                   IF #Minuty < 10 THEN
                       #StrMin := CONCAT(IN1 := '0', IN2 := #StrMin);
                   END_IF;
                   IF #Sekundy < 10 THEN
                       #StrSec := CONCAT(IN1 := '0', IN2 := #StrSec);
                   END_IF;

                   IF "DB_Data".Stanowisko1."Time".RemainingSec <= 0 AND "DB_Data".Stanowisko1."Time".Blink THEN
                       "DB_Data".Stanowisko1."Time".RemainingStr := '     ';
                   ELSE
                       "DB_Data".Stanowisko1."Time".RemainingStr := CONCAT(IN1 := #StrMin, IN2 := CONCAT(IN1 := ':', IN2 := #StrSec));
                   END_IF;

           END_CASE;

           //Przejscie do stanu awarii
           IF "DB_Data".Stanowisko1.Commands.ReportFault.State THEN
               "DB_Data".Stanowisko1.Production.State := 3;
               "DB_Data".Stanowisko1.Commands.ReportFault.State := 0;
           END_IF;

           //Przejscie do zakonczenia montazu
           IF "DB_Data".Stanowisko1.Commands.FInish.State THEN
               "DB_Data".Stanowisko1.Production.State := 2;
               "DB_Data".Stanowisko1.Commands.FInish.State := 0;
           END_IF;

       2:
           //Ustawienie przycisków
           "DB_Data".Stanowisko1.Commands.Start.Enable := 0;
           "DB_Data".Stanowisko1.Commands.AbortProcess.Enable := 0;
           "DB_Data".Stanowisko1.Commands.FInish.Enable := 0;
           "DB_Data".Stanowisko1.Commands.ReportFault.Enable := 0;

           #temp_start_time := RD_LOC_T(OUT => "DB_Zlecenia".NastepneZlecenie.Zlecenie."Time".Stanowisko1.EndTime); // Zapis czasu zakonczenia

           //Funkcja zapisujaca wyrob do bazy danych dla innych stanowisk
           FOR #i := 0 TO 199 DO

               // szukanie pierwszego wolnego miejsca (czyli takiego, gdzie ID zlecenia to 0)
               IF "DB_Zlecenia".Zlecenie[#i].Zlecenie.ID = 0 THEN

                   "DB_Zlecenia".Zlecenie[#i] := "DB_Zlecenia".NastepneZlecenie;

                   //Status stanowiska 1 - praca zakonczona
                   "DB_Zlecenia".Zlecenie[#i].Zlecenie.Status[0] := TRUE;

                   //Obliczenie faktycznego czasu pracy (sekundy, zaokraglone)
                   #temp_diff_time := "DB_Zlecenia".Zlecenie[#i].Zlecenie."Time".Stanowisko1.EndTime - "DB_Zlecenia".Zlecenie[#i].Zlecenie."Time".Stanowisko1.StartTime;
                   "DB_Zlecenia".Zlecenie[#i].Zlecenie."Time".Stanowisko1.ActualTime := DINT_TO_INT((TIME_TO_DINT(#temp_diff_time) + 500) / 1000);

                   //Jesli zlecenie mialo wiecej niz 1 sztuke - zostaw ID/Model, zmniejsz PartNo, wyczysc Time/Alarm
                   IF "DB_Zlecenia".NastepneZlecenie.Zlecenie.PartNo > 1 THEN
                       "DB_Zlecenia".NastepneZlecenie.Zlecenie.PartNo := "DB_Zlecenia".NastepneZlecenie.Zlecenie.PartNo - 1;
                       "DB_Zlecenia".NastepneZlecenie.Zlecenie."Time" := "DB_Zlecenia".PusteZlecenie.Zlecenie."Time";
                       "DB_Zlecenia".NastepneZlecenie.Zlecenie.Alarm := "DB_Zlecenia".PusteZlecenie.Zlecenie.Alarm;
                   ELSE
                       "DB_Zlecenia".NastepneZlecenie := "DB_Zlecenia".PusteZlecenie;
                   END_IF;
                   EXIT;
               END_IF;
           END_FOR;

           "DB_Data".Stanowisko1.Stats.DoneToday := "DB_Data".Stanowisko1.Stats.DoneToday + 1;
           "DB_Data".DoneAllTime[0] := "DB_Data".DoneAllTime[0] + 1;

           "DB_Data".Stanowisko1.Production.State := 0;
       3:
           //Ustawienie przycisków
           "DB_Data".Stanowisko1.Commands.Start.Enable := 0;
           "DB_Data".Stanowisko1.Commands.AbortProcess.Enable := 1;
           "DB_Data".Stanowisko1.Commands.FInish.Enable := 0;
           "DB_Data".Stanowisko1.Commands.ReportFault.Enable := 0;

           //Dodanie alarmow
           "DB_Zlecenia".NastepneZlecenie.Zlecenie.Alarm.Stanowisko1 := "DB_Data".Stanowisko1.Commands.FaultReason;

           IF "DB_Data".Stanowisko1.Commands.AbortProcess.State THEN
               #temp_start_time := RD_LOC_T(OUT => "DB_Zlecenia".NastepneZlecenie.Zlecenie."Time".Stanowisko1.EndTime); // Zapis czasu zakonczenia

               //Funkcja zapisujaca wyrob do bazy danych dla innych stanowisk
               FOR #i := 0 TO 199 DO
                   IF "DB_Zlecenia".Zlecenie[#i].Zlecenie.ID = 0 THEN

                       "DB_Zlecenia".Zlecenie[#i] := "DB_Zlecenia".NastepneZlecenie;
                       "DB_Zlecenia".Zlecenie[#i].Zlecenie."Time".Stanowisko1.Abort := TRUE;

                       //Status stanowiska 1 - praca zakonczona (przez abort)
                       "DB_Zlecenia".Zlecenie[#i].Zlecenie.Status[0] := TRUE;

                       //Obliczenie faktycznego czasu pracy (sekundy, zaokraglone)
                       #temp_diff_time := "DB_Zlecenia".Zlecenie[#i].Zlecenie."Time".Stanowisko1.EndTime - "DB_Zlecenia".Zlecenie[#i].Zlecenie."Time".Stanowisko1.StartTime;
                       "DB_Zlecenia".Zlecenie[#i].Zlecenie."Time".Stanowisko1.ActualTime := DINT_TO_INT((TIME_TO_DINT(#temp_diff_time) + 500) / 1000);

                       IF "DB_Zlecenia".NastepneZlecenie.Zlecenie.PartNo > 1 THEN
                           "DB_Zlecenia".NastepneZlecenie.Zlecenie.PartNo := "DB_Zlecenia".NastepneZlecenie.Zlecenie.PartNo - 1;
                           "DB_Zlecenia".NastepneZlecenie.Zlecenie."Time" := "DB_Zlecenia".PusteZlecenie.Zlecenie."Time";
                           "DB_Zlecenia".NastepneZlecenie.Zlecenie.Alarm := "DB_Zlecenia".PusteZlecenie.Zlecenie.Alarm;
                       ELSE
                           "DB_Zlecenia".NastepneZlecenie := "DB_Zlecenia".PusteZlecenie;
                       END_IF;

                       "DB_Data".Stanowisko1.Commands.AbortProcess.State := 0;
                       "DB_Data".Stanowisko1.Production.State := 0;
                       EXIT;
                   END_IF;
               END_FOR;
           END_IF;

   END_CASE;
   IF "DB_Data".Stanowisko1.Commands.AbortProcess.State THEN
       "DB_Data".Stanowisko1.Production.State := 0;
       "DB_Data".Stanowisko1.Commands.AbortProcess.State := 0;

       #temp_start_time := RD_LOC_T(OUT => "DB_Zlecenia".NastepneZlecenie.Zlecenie."Time".Stanowisko1.EndTime); // Zapis czasu zakonczenia

       //Funkcja zapisujaca wyrob do bazy danych dla innych stanowisk
       FOR #i := 0 TO 199 DO
           IF "DB_Zlecenia".Zlecenie[#i].Zlecenie.ID = 0 THEN

               "DB_Zlecenia".Zlecenie[#i] := "DB_Zlecenia".NastepneZlecenie;
               "DB_Zlecenia".Zlecenie[#i].Zlecenie."Time".Stanowisko1.Abort := TRUE;

               //Status stanowiska 1 - praca zakonczona (przez abort)
               "DB_Zlecenia".Zlecenie[#i].Zlecenie.Status[0] := TRUE;

               //Obliczenie faktycznego czasu pracy (sekundy, zaokraglone)
               #temp_diff_time := "DB_Zlecenia".Zlecenie[#i].Zlecenie."Time".Stanowisko1.EndTime - "DB_Zlecenia".Zlecenie[#i].Zlecenie."Time".Stanowisko1.StartTime;
               "DB_Zlecenia".Zlecenie[#i].Zlecenie."Time".Stanowisko1.ActualTime := DINT_TO_INT((TIME_TO_DINT(#temp_diff_time) + 500) / 1000);

               IF "DB_Zlecenia".NastepneZlecenie.Zlecenie.PartNo > 1 THEN
                   "DB_Zlecenia".NastepneZlecenie.Zlecenie.PartNo := "DB_Zlecenia".NastepneZlecenie.Zlecenie.PartNo - 1;
                   "DB_Zlecenia".NastepneZlecenie.Zlecenie."Time" := "DB_Zlecenia".PusteZlecenie.Zlecenie."Time";
                   "DB_Zlecenia".NastepneZlecenie.Zlecenie.Alarm := "DB_Zlecenia".PusteZlecenie.Zlecenie.Alarm;
               ELSE
                   "DB_Zlecenia".NastepneZlecenie := "DB_Zlecenia".PusteZlecenie;
               END_IF;

               "DB_Data".Stanowisko1.Commands.AbortProcess.State := 0;
               "DB_Data".Stanowisko1.Production.State := 0;
               EXIT;
           END_IF;
       END_FOR;
   END_IF;
   IF "DB_Data".Stanowisko1.HMI.Clear THEN
       "DB_Data".Stanowisko1.Stats.DoneToday := 0;
       "DB_Data".Stanowisko1.HMI.Clear := 0;
   END_IF;
END_ORGANIZATION_BLOCK

ORGANIZATION_BLOCK "Czujniki"   // OB124, SCL, ProgramCycle
TITLE = "Main Program Sweep (Cycle)"
{ S7_Optimized_Access := 'TRUE' }
VERSION : 0.1
   VAR_INPUT
      Initial_Call : Bool;   // Initial call of this OB
      Remanence : Bool;   // =True, if remanent data are available
   END_VAR
   VAR_TEMP
      i : Int;
   END_VAR
BEGIN
   // ------------------------------------------------------------------
   // 1. PRZEKAZANIE DANYCH DO APLIKACJI C# / SQL
   // ------------------------------------------------------------------
   //Czujniki odleglosciowe od 1 stanowiska do 4
   "DB_Data".Stanowisko1.Sensors.PalletPresent := "Tag_1";
   "DB_Data".Stanowisko2.Sensors.PalletPresent := "Tag_2";
   "DB_Data".Stanowisko3.Sensors.PalletPresent := "Tag_10";
   "DB_Data".StanowiskoQC.Sensors.PalletPresent := "Tag_11";

   // Zapisujemy do bazy, czy czytnik w ogóle widzi tag (z fizycznego wejścia)
   "DB_Data".Stanowisko1.Sensors.RFID.TagPresent := "RFID1";
   "DB_Data".Stanowisko2.Sensors.RFID.TagPresent := "RFID2";
   "DB_Data".Stanowisko3.Sensors.RFID.TagPresent := "RFID3";
   "DB_Data".StanowiskoQC.Sensors.RFID.TagPresent := "RFID4";


   FOR #i := 1 TO 9 DO
       "DB_PTL".PTL_state[#i - 1] := "DB_PTL".PTL_Buttons[#i].%X0;
   END_FOR;

   FOR #i := 0 TO 8 DO
       IF "DB_PTL".PTL_state[#i] AND NOT "DB_PTL".PTL_State_Old[#i] THEN

           CASE #i OF
               0..2:
                   //Stanowisko1 - kontenery 1..3 (przyciski 0..2)
                   IF "DB_Data".Stanowisko1.HMI.Container[#i + 1].value > 0 THEN
                       "DB_Data".Stanowisko1.HMI.Container[#i + 1].value -= 1;
                   END_IF;

               3..5:
                   //Stanowisko2 - kontenery 1..3 (przyciski 3..5)
                   IF "DB_Data".Stanowisko2.HMI.Container[#i - 2].value > 0 THEN
                       "DB_Data".Stanowisko2.HMI.Container[#i - 2].value -= 1;
                   END_IF;

               6..8:
                   //Stanowisko3 - kontenery 1..3 (przyciski 6..8)
                   IF "DB_Data".Stanowisko3.HMI.Container[#i - 5].value > 0 THEN
                       "DB_Data".Stanowisko3.HMI.Container[#i - 5].value -= 1;
                   END_IF;

           END_CASE;

       END_IF;

       // zapamiętaj stan na następny cykl (zawsze, na końcu)
       "DB_PTL".PTL_State_Old[#i] := "DB_PTL".PTL_state[#i];
   END_FOR;


   // 1. Inicjalizacja parametrów połączenia
   IF NOT "DB_PTL".InitDone THEN
       "DB_PTL".ConnParams.InterfaceId := 64;
       "DB_PTL".ConnParams.ID := 1;
       "DB_PTL".ConnParams.ConnectionType := 11;
       "DB_PTL".ConnParams.ActiveEstablished := TRUE;
       "DB_PTL".ConnParams.RemoteAddress.ADDR[1] := 192;
       "DB_PTL".ConnParams.RemoteAddress.ADDR[2] := 168;
       "DB_PTL".ConnParams.RemoteAddress.ADDR[3] := 1;
       "DB_PTL".ConnParams.RemoteAddress.ADDR[4] := 30;
       "DB_PTL".ConnParams.RemotePort := 502;
       "DB_PTL".Wyzwalacz := TRUE;

       "DB_PTL".InitDone := TRUE;
   END_IF;

   // 2. Wywołanie bloku Modbus Client do odczytu PTL Node 1
   "MB_CLIENT_DB"(
                  REQ := "DB_PTL".Wyzwalacz,
                  DISCONNECT := FALSE,
                  MB_MODE := 0,
                  MB_DATA_ADDR := 40017,                   // Zaczynamy czytać od rejestru 17...
                  MB_DATA_LEN := 9,                       // ...i czytamy od razu 9 rejestrów naraz!
                  DONE => "DB_PTL".mb_done,
                  BUSY => "DB_PTL".mb_busy,
                  ERROR => "DB_PTL".mb_error,
                  STATUS => "DB_PTL".mb_status,
                  CONNECT := "DB_PTL".ConnParams,
                  MB_DATA_PTR := "DB_PTL".PTL_Buttons     // Wrzucamy wszystko do naszej tablicy
   );
END_ORGANIZATION_BLOCK

ORGANIZATION_BLOCK "Kontenery"   // OB125, SCL, ProgramCycle
TITLE = "Main Program Sweep (Cycle)"
{ S7_Optimized_Access := 'TRUE' }
VERSION : 0.1
   VAR_INPUT
      Initial_Call : Bool;   // Initial call of this OB
      Remanence : Bool;   // =True, if remanent data are available
   END_VAR
BEGIN
   // ==========================================================================
   // Stanowisko 1
   // ==========================================================================
   //Tor 1
   IF "DB_Data".Stanowisko1.HMI.Container[1].value = 0 THEN
       "DB_Data".Stanowisko1.HMI.Container[1].Subtract.Enable := FALSE;
       "DB_Data".Stanowisko1.HMI.Container[1].Add.Enable := TRUE;
   END_IF;
   IF "DB_Data".Stanowisko1.HMI.Container[1].value = 1 OR "DB_Data".Stanowisko1.HMI.Container[1].value = 2 THEN
       "DB_Data".Stanowisko1.HMI.Container[1].Subtract.Enable := TRUE;
       "DB_Data".Stanowisko1.HMI.Container[1].Add.Enable := TRUE;
   END_IF;
   IF "DB_Data".Stanowisko1.HMI.Container[1].value = 3 THEN
       "DB_Data".Stanowisko1.HMI.Container[1].Add.Enable := FALSE;
   END_IF;
   IF "DB_Data".Stanowisko1.HMI.Container[1].Subtract.Status THEN
       "DB_Data".Stanowisko1.HMI.Container[1].value -= 1;
       "DB_Data".Stanowisko1.HMI.Container[1].Subtract.Status := FALSE;
   END_IF;
   IF "DB_Data".Stanowisko1.HMI.Container[1].Add.Status THEN
       "DB_Data".Stanowisko1.HMI.Container[1].value += 1;
       "DB_Data".Stanowisko1.HMI.Container[1].Add.Status := FALSE;
   END_IF;

   //Tor 2
   IF "DB_Data".Stanowisko1.HMI.Container[2].value = 0 THEN
       "DB_Data".Stanowisko1.HMI.Container[2].Subtract.Enable := FALSE;
       "DB_Data".Stanowisko1.HMI.Container[2].Add.Enable := TRUE;
   END_IF;
   IF "DB_Data".Stanowisko1.HMI.Container[2].value = 1 OR "DB_Data".Stanowisko1.HMI.Container[2].value = 2 THEN
       "DB_Data".Stanowisko1.HMI.Container[2].Subtract.Enable := TRUE;
       "DB_Data".Stanowisko1.HMI.Container[2].Add.Enable := TRUE;
   END_IF;
   IF "DB_Data".Stanowisko1.HMI.Container[2].value = 3 THEN
       "DB_Data".Stanowisko1.HMI.Container[2].Add.Enable := FALSE;
   END_IF;
   IF "DB_Data".Stanowisko1.HMI.Container[2].Subtract.Status THEN
       "DB_Data".Stanowisko1.HMI.Container[2].value -= 1;
       "DB_Data".Stanowisko1.HMI.Container[2].Subtract.Status := FALSE;
   END_IF;
   IF "DB_Data".Stanowisko1.HMI.Container[2].Add.Status THEN
       "DB_Data".Stanowisko1.HMI.Container[2].value += 1;
       "DB_Data".Stanowisko1.HMI.Container[2].Add.Status := FALSE;
   END_IF;

   //Tor 3
   IF "DB_Data".Stanowisko1.HMI.Container[3].value = 0 THEN
       "DB_Data".Stanowisko1.HMI.Container[3].Subtract.Enable := FALSE;
       "DB_Data".Stanowisko1.HMI.Container[3].Add.Enable := TRUE;
   END_IF;
   IF "DB_Data".Stanowisko1.HMI.Container[3].value = 1 OR "DB_Data".Stanowisko1.HMI.Container[3].value = 2 THEN
       "DB_Data".Stanowisko1.HMI.Container[3].Subtract.Enable := TRUE;
       "DB_Data".Stanowisko1.HMI.Container[3].Add.Enable := TRUE;
   END_IF;
   IF "DB_Data".Stanowisko1.HMI.Container[3].value = 3 THEN
       "DB_Data".Stanowisko1.HMI.Container[3].Add.Enable := FALSE;
   END_IF;
   IF "DB_Data".Stanowisko1.HMI.Container[3].Subtract.Status THEN
       "DB_Data".Stanowisko1.HMI.Container[3].value -= 1;
       "DB_Data".Stanowisko1.HMI.Container[3].Subtract.Status := FALSE;
   END_IF;
   IF "DB_Data".Stanowisko1.HMI.Container[3].Add.Status THEN
       "DB_Data".Stanowisko1.HMI.Container[3].value += 1;
       "DB_Data".Stanowisko1.HMI.Container[3].Add.Status := FALSE;
   END_IF;

   // ==========================================================================
   // Stanowisko 2
   // ==========================================================================
   //Tor 1
   IF "DB_Data".Stanowisko2.HMI.Container[1].value = 0 THEN
       "DB_Data".Stanowisko2.HMI.Container[1].Subtract.Enable := FALSE;
       "DB_Data".Stanowisko2.HMI.Container[1].Add.Enable := TRUE;
   END_IF;
   IF "DB_Data".Stanowisko2.HMI.Container[1].value = 1 OR "DB_Data".Stanowisko2.HMI.Container[1].value = 2 THEN
       "DB_Data".Stanowisko2.HMI.Container[1].Subtract.Enable := TRUE;
       "DB_Data".Stanowisko2.HMI.Container[1].Add.Enable := TRUE;
   END_IF;
   IF "DB_Data".Stanowisko2.HMI.Container[1].value = 3 THEN
       "DB_Data".Stanowisko2.HMI.Container[1].Add.Enable := FALSE;
   END_IF;
   IF "DB_Data".Stanowisko2.HMI.Container[1].Subtract.Status THEN
       "DB_Data".Stanowisko2.HMI.Container[1].value -= 1;
       "DB_Data".Stanowisko2.HMI.Container[1].Subtract.Status := FALSE;
   END_IF;
   IF "DB_Data".Stanowisko2.HMI.Container[1].Add.Status THEN
       "DB_Data".Stanowisko2.HMI.Container[1].value += 1;
       "DB_Data".Stanowisko2.HMI.Container[1].Add.Status := FALSE;
   END_IF;

   //Tor 2
   IF "DB_Data".Stanowisko2.HMI.Container[2].value = 0 THEN
       "DB_Data".Stanowisko2.HMI.Container[2].Subtract.Enable := FALSE;
       "DB_Data".Stanowisko2.HMI.Container[2].Add.Enable := TRUE;
   END_IF;
   IF "DB_Data".Stanowisko2.HMI.Container[2].value = 1 OR "DB_Data".Stanowisko2.HMI.Container[2].value = 2 THEN
       "DB_Data".Stanowisko2.HMI.Container[2].Subtract.Enable := TRUE;
       "DB_Data".Stanowisko2.HMI.Container[2].Add.Enable := TRUE;
   END_IF;
   IF "DB_Data".Stanowisko2.HMI.Container[2].value = 3 THEN
       "DB_Data".Stanowisko2.HMI.Container[2].Add.Enable := FALSE;
   END_IF;
   IF "DB_Data".Stanowisko2.HMI.Container[2].Subtract.Status THEN
       "DB_Data".Stanowisko2.HMI.Container[2].value -= 1;
       "DB_Data".Stanowisko2.HMI.Container[2].Subtract.Status := FALSE;
   END_IF;
   IF "DB_Data".Stanowisko2.HMI.Container[2].Add.Status THEN
       "DB_Data".Stanowisko2.HMI.Container[2].value += 1;
       "DB_Data".Stanowisko2.HMI.Container[2].Add.Status := FALSE;
   END_IF;

   //Tor 3
   IF "DB_Data".Stanowisko2.HMI.Container[3].value = 0 THEN
       "DB_Data".Stanowisko2.HMI.Container[3].Subtract.Enable := FALSE;
       "DB_Data".Stanowisko2.HMI.Container[3].Add.Enable := TRUE;
   END_IF;
   IF "DB_Data".Stanowisko2.HMI.Container[3].value = 1 OR "DB_Data".Stanowisko2.HMI.Container[3].value = 2 THEN
       "DB_Data".Stanowisko2.HMI.Container[3].Subtract.Enable := TRUE;
       "DB_Data".Stanowisko2.HMI.Container[3].Add.Enable := TRUE;
   END_IF;
   IF "DB_Data".Stanowisko2.HMI.Container[3].value = 3 THEN
       "DB_Data".Stanowisko2.HMI.Container[3].Add.Enable := FALSE;
   END_IF;
   IF "DB_Data".Stanowisko2.HMI.Container[3].Subtract.Status THEN
       "DB_Data".Stanowisko2.HMI.Container[3].value -= 1;
       "DB_Data".Stanowisko2.HMI.Container[3].Subtract.Status := FALSE;
   END_IF;
   IF "DB_Data".Stanowisko2.HMI.Container[3].Add.Status THEN
       "DB_Data".Stanowisko2.HMI.Container[3].value += 1;
       "DB_Data".Stanowisko2.HMI.Container[3].Add.Status := FALSE;
   END_IF;

   // ==========================================================================
   // Stanowisko 3
   // ==========================================================================
   //Tor 1
   IF "DB_Data".Stanowisko3.HMI.Container[1].value = 0 THEN
       "DB_Data".Stanowisko3.HMI.Container[1].Subtract.Enable := FALSE;
       "DB_Data".Stanowisko3.HMI.Container[1].Add.Enable := TRUE;
   END_IF;
   IF "DB_Data".Stanowisko3.HMI.Container[1].value = 1 OR "DB_Data".Stanowisko3.HMI.Container[1].value = 2 THEN
       "DB_Data".Stanowisko3.HMI.Container[1].Subtract.Enable := TRUE;
       "DB_Data".Stanowisko3.HMI.Container[1].Add.Enable := TRUE;
   END_IF;
   IF "DB_Data".Stanowisko3.HMI.Container[1].value = 3 THEN
       "DB_Data".Stanowisko3.HMI.Container[1].Add.Enable := FALSE;
   END_IF;
   IF "DB_Data".Stanowisko3.HMI.Container[1].Subtract.Status THEN
       "DB_Data".Stanowisko3.HMI.Container[1].value -= 1;
       "DB_Data".Stanowisko3.HMI.Container[1].Subtract.Status := FALSE;
   END_IF;
   IF "DB_Data".Stanowisko3.HMI.Container[1].Add.Status THEN
       "DB_Data".Stanowisko3.HMI.Container[1].value += 1;
       "DB_Data".Stanowisko3.HMI.Container[1].Add.Status := FALSE;
   END_IF;

   //Tor 2
   IF "DB_Data".Stanowisko3.HMI.Container[2].value = 0 THEN
       "DB_Data".Stanowisko3.HMI.Container[2].Subtract.Enable := FALSE;
       "DB_Data".Stanowisko3.HMI.Container[2].Add.Enable := TRUE;
   END_IF;
   IF "DB_Data".Stanowisko3.HMI.Container[2].value = 1 OR "DB_Data".Stanowisko3.HMI.Container[2].value = 2 THEN
       "DB_Data".Stanowisko3.HMI.Container[2].Subtract.Enable := TRUE;
       "DB_Data".Stanowisko3.HMI.Container[2].Add.Enable := TRUE;
   END_IF;
   IF "DB_Data".Stanowisko3.HMI.Container[2].value = 3 THEN
       "DB_Data".Stanowisko3.HMI.Container[2].Add.Enable := FALSE;
   END_IF;
   IF "DB_Data".Stanowisko3.HMI.Container[2].Subtract.Status THEN
       "DB_Data".Stanowisko3.HMI.Container[2].value -= 1;
       "DB_Data".Stanowisko3.HMI.Container[2].Subtract.Status := FALSE;
   END_IF;
   IF "DB_Data".Stanowisko3.HMI.Container[2].Add.Status THEN
       "DB_Data".Stanowisko3.HMI.Container[2].value += 1;
       "DB_Data".Stanowisko3.HMI.Container[2].Add.Status := FALSE;
   END_IF;

   //Tor 3
   IF "DB_Data".Stanowisko3.HMI.Container[3].value = 0 THEN
       "DB_Data".Stanowisko3.HMI.Container[3].Subtract.Enable := FALSE;
       "DB_Data".Stanowisko3.HMI.Container[3].Add.Enable := TRUE;
   END_IF;
   IF "DB_Data".Stanowisko3.HMI.Container[3].value = 1 OR "DB_Data".Stanowisko3.HMI.Container[3].value = 2 THEN
       "DB_Data".Stanowisko3.HMI.Container[3].Subtract.Enable := TRUE;
       "DB_Data".Stanowisko3.HMI.Container[3].Add.Enable := TRUE;
   END_IF;
   IF "DB_Data".Stanowisko3.HMI.Container[3].value = 3 THEN
       "DB_Data".Stanowisko3.HMI.Container[3].Add.Enable := FALSE;
   END_IF;
   IF "DB_Data".Stanowisko3.HMI.Container[3].Subtract.Status THEN
       "DB_Data".Stanowisko3.HMI.Container[3].value -= 1;
       "DB_Data".Stanowisko3.HMI.Container[3].Subtract.Status := FALSE;
   END_IF;
   IF "DB_Data".Stanowisko3.HMI.Container[3].Add.Status THEN
       "DB_Data".Stanowisko3.HMI.Container[3].value += 1;
       "DB_Data".Stanowisko3.HMI.Container[3].Add.Status := FALSE;
   END_IF;
END_ORGANIZATION_BLOCK

ORGANIZATION_BLOCK "Stanowisko2"   // OB126, SCL, ProgramCycle
TITLE = "Main Program Sweep (Cycle)"
{ S7_Optimized_Access := 'TRUE' }
VERSION : 0.1
   VAR_INPUT
      Initial_Call : Bool;   // Initial call of this OB
      Remanence : Bool;   // =True, if remanent data are available
   END_VAR
   VAR_TEMP
      temp_start_time : Int;
      temp_taget_time : Int;
      i : Int;
      Czas_DTL : DTL;
      Status_Czasu : Int;
      Minuty : Int;
      Sekundy : Int;
      StrMin : String;
      StrSec : String;
      temp_diff_time : Time;
   END_VAR
BEGIN
   // ===================== STANOWISKO 2 =====================
   CASE "DB_Data".Stanowisko2.Production.State OF

       0:
           //Ustawienie przyciskow
           "DB_Data".Stanowisko2.Commands.AbortProcess.Enable := 0;
           "DB_Data".Stanowisko2.Commands.FInish.Enable := 0;
           "DB_Data".Stanowisko2.Commands.ReportFault.Enable := 0;

           //Wyzerowanie stanu przyciskow (na wypadek zaleglych klikniec)
           "DB_Data".Stanowisko2.Commands.FInish.State := 0;
           "DB_Data".Stanowisko2.Commands.ReportFault.State := 0;

           //Ustawienie awarii na 0
           "DB_Data".Stanowisko2.Commands.FaultReason.DamagedPart := 0;
           "DB_Data".Stanowisko2.Commands.FaultReason.MissingPart := 0;
           "DB_Data".Stanowisko2.Commands.FaultReason.Other := 0;
           "DB_Data".Stanowisko2.Commands.FaultReason.PalletFault := 0;
           "DB_Data".Stanowisko2.Commands.FaultReason.SensorFault := 0;
           "DB_Data".Stanowisko2.Commands.FaultReason.WrongInstruction := 0;

           //Reset czasu cyklu na wyswietlaczu
           "DB_Data".Stanowisko2."Time".RemainingStr := '00:00';

           //Reset numeru zlecenia
           "DB_Data".Stanowisko2.Production.OrderNo := 0;
           "DB_Data".Stanowisko2.Production.ProductNo := 0;

           //Zerowanie flagi ladowania
           "DB_Data".Stanowisko2.Stats.Loaded := 0;

           "DB_Data".Stanowisko2.Stats.Instruction := 1;

           //Zabezpieczenie indeksu bazy (ustawienie na wartość pustą)
           "DB_Data".ZlecenieIndex[1] := -1;
           "RFID_test".Bufor_Odczyt2[0] := 0;
           "RFID_test".Bufor_Odczyt2[1] := 0;
           "RFID_test".Bufor_Odczyt2[2] := 0;

           //Przejscie do montazu jezeli paletka jest aktywna i start klikniety
           IF "DB_Data".Stanowisko2.Sensors.PalletPresent THEN
               "DB_Data".Stanowisko2.Commands.Start.Enable := 1;
               IF "DB_Data".Stanowisko2.Commands.Start.State THEN
                   "DB_Data".Stanowisko2.Production.State := 1;
                   "DB_Data".Stanowisko2.Commands.Start.State := 0;
                   "DB_Data".Stanowisko2.MontazState := 0;
               END_IF;
           ELSE
               "DB_Data".Stanowisko2.Commands.Start.Enable := 0;
           END_IF;


       1:
           //Ustawienie przycisków
           "DB_Data".Stanowisko2.Commands.Start.Enable := 0;
           "DB_Data".Stanowisko2.Commands.AbortProcess.Enable := 1;
           "DB_Data".Stanowisko2.Commands.FInish.Enable := 1;
           "DB_Data".Stanowisko2.Commands.ReportFault.Enable := 1;

           CASE "DB_Data".Stanowisko2.MontazState OF
               0:
                   // Wysłanie komendy odczytu
                   "DB_Data".Stanowisko2.Sensors.RFID.CmdRead := TRUE;

                   // Pobranie danych z bufora
                   "DB_Data".Stanowisko2.Production.OrderNo := BYTE_TO_INT("RFID_test".Bufor_Odczyt2[0]);
                   "DB_Data".Stanowisko2.Stats.Instruction := BYTE_TO_INT("RFID_test".Bufor_Odczyt2[1]);
                   "DB_Data".Stanowisko2.Production.ProductNo := BYTE_TO_INT("RFID_test".Bufor_Odczyt2[2]);

                   // Szukanie TargetTime w tablicy zleceń
                   FOR #i := 0 TO 199 DO
                       IF "DB_Zlecenia".Zlecenie[#i].Zlecenie.ID = "DB_Data".Stanowisko2.Production.OrderNo AND "DB_Zlecenia".Zlecenie[#i].Zlecenie.PartNo = "DB_Data".Stanowisko2.Production.ProductNo THEN
                           "DB_Data".Stanowisko2."Time".RemainingSec := "DB_Zlecenia".Zlecenie[#i].Zlecenie."Time".Stanowisko2.TargetTime;
                           "DB_Data".ZlecenieIndex[1] := #i;
                           EXIT;
                       END_IF;
                   END_FOR;

                   IF "DB_Data".Stanowisko2.Production.OrderNo <> 0 THEN
                       "DB_Data".Stanowisko2.MontazState := 1;
                   END_IF;

               1:
                   "DB_Data".Stanowisko2."Time".Blink := FALSE;
                   "DB_Data".Stanowisko2.Sensors.RFID.CmdRead := FALSE;
                   #temp_start_time := RD_LOC_T(OUT => "DB_Zlecenia".Zlecenie["DB_Data".ZlecenieIndex[1]].Zlecenie."Time".Stanowisko2.StartTime);

                   "DB_Data".Stanowisko2.MontazState := 2;

               2:
                   #Status_Czasu := RD_SYS_T(OUT => #Czas_DTL);

                   IF #Czas_DTL.SECOND <> "DB_Data".Stanowisko2."Time".LastSec THEN
                       "DB_Data".Stanowisko2."Time".LastSec := #Czas_DTL.SECOND;

                       IF "DB_Data".Stanowisko2."Time".RemainingSec > 0 THEN
                           "DB_Data".Stanowisko2."Time".RemainingSec := "DB_Data".Stanowisko2."Time".RemainingSec - 1;
                       END_IF;

                       IF "DB_Data".Stanowisko2."Time".RemainingSec <= 0 THEN
                           "DB_Data".Stanowisko2."Time".Blink := NOT "DB_Data".Stanowisko2."Time".Blink;
                       END_IF;
                   END_IF;

                   #Minuty := "DB_Data".Stanowisko2."Time".RemainingSec / 60;
                   #Sekundy := "DB_Data".Stanowisko2."Time".RemainingSec MOD 60;

                   #StrMin := INT_TO_STRING(#Minuty);
                   #StrSec := INT_TO_STRING(#Sekundy);

                   #StrMin := RIGHT(IN := #StrMin, L := LEN(#StrMin) - 1);
                   #StrSec := RIGHT(IN := #StrSec, L := LEN(#StrSec) - 1);

                   IF #Minuty < 10 THEN
                       #StrMin := CONCAT(IN1 := '0', IN2 := #StrMin);
                   END_IF;
                   IF #Sekundy < 10 THEN
                       #StrSec := CONCAT(IN1 := '0', IN2 := #StrSec);
                   END_IF;

                   IF "DB_Data".Stanowisko2."Time".RemainingSec <= 0 AND "DB_Data".Stanowisko2."Time".Blink THEN
                       "DB_Data".Stanowisko2."Time".RemainingStr := '     ';
                   ELSE
                       "DB_Data".Stanowisko2."Time".RemainingStr := CONCAT(IN1 := #StrMin, IN2 := CONCAT(IN1 := ':', IN2 := #StrSec));
                   END_IF;

           END_CASE;

           //Przejscie do stanu awarii
           IF "DB_Data".Stanowisko2.Commands.ReportFault.State THEN
               "DB_Data".Stanowisko2.Production.State := 3;
               "DB_Data".Stanowisko2.Commands.ReportFault.State := 0;
           END_IF;

           //Przejscie do zakonczenia montazu
           IF "DB_Data".Stanowisko2.Commands.FInish.State THEN
               "DB_Data".Stanowisko2.Production.State := 2;
               "DB_Data".Stanowisko2.Commands.FInish.State := 0;
           END_IF;

       2:
           "DB_Data".Stanowisko2.Commands.Start.Enable := 0;
           "DB_Data".Stanowisko2.Commands.AbortProcess.Enable := 0;
           "DB_Data".Stanowisko2.Commands.FInish.Enable := 0;
           "DB_Data".Stanowisko2.Commands.ReportFault.Enable := 0;

           // Zapis tylko jeśli indeks został znaleziony
           IF "DB_Data".ZlecenieIndex[1] >= 0 THEN
               #temp_start_time := RD_LOC_T(OUT => "DB_Zlecenia".Zlecenie["DB_Data".ZlecenieIndex[1]].Zlecenie."Time".Stanowisko2.EndTime);

               //Status stanowiska 2 - praca zakonczona
               "DB_Zlecenia".Zlecenie["DB_Data".ZlecenieIndex[1]].Zlecenie.Status[1] := TRUE;

               //Obliczenie faktycznego czasu pracy (sekundy, zaokraglone)
               #temp_diff_time := "DB_Zlecenia".Zlecenie["DB_Data".ZlecenieIndex[1]].Zlecenie."Time".Stanowisko2.EndTime - "DB_Zlecenia".Zlecenie["DB_Data".ZlecenieIndex[1]].Zlecenie."Time".Stanowisko2.StartTime;
               "DB_Zlecenia".Zlecenie["DB_Data".ZlecenieIndex[1]].Zlecenie."Time".Stanowisko2.ActualTime := DINT_TO_INT((TIME_TO_DINT(#temp_diff_time) + 500) / 1000);
           END_IF;

           "DB_Data".Stanowisko2.Stats.DoneToday := "DB_Data".Stanowisko2.Stats.DoneToday + 1;
           "DB_Data".DoneAllTime[1] := "DB_Data".DoneAllTime[1] + 1;

           "DB_Data".ZlecenieIndex[1] := -1;
           "DB_Data".Stanowisko2.Production.State := 0;

       3:
           "DB_Data".Stanowisko2.Commands.Start.Enable := 0;
           "DB_Data".Stanowisko2.Commands.AbortProcess.Enable := 1;
           "DB_Data".Stanowisko2.Commands.FInish.Enable := 0;
           "DB_Data".Stanowisko2.Commands.ReportFault.Enable := 0;

           IF "DB_Data".ZlecenieIndex[1] >= 0 THEN
               "DB_Zlecenia".Zlecenie["DB_Data".ZlecenieIndex[1]].Zlecenie.Alarm.Stanowisko2 := "DB_Data".Stanowisko2.Commands.FaultReason;
           END_IF;

           IF "DB_Data".Stanowisko2.Commands.AbortProcess.State THEN
               IF "DB_Data".ZlecenieIndex[1] >= 0 THEN
                   #temp_start_time := RD_LOC_T(OUT => "DB_Zlecenia".Zlecenie["DB_Data".ZlecenieIndex[1]].Zlecenie."Time".Stanowisko2.EndTime);
                   "DB_Zlecenia".Zlecenie["DB_Data".ZlecenieIndex[1]].Zlecenie."Time".Stanowisko2.Abort := TRUE;

                   //Status stanowiska 2 - praca zakonczona (przez abort)
                   "DB_Zlecenia".Zlecenie["DB_Data".ZlecenieIndex[1]].Zlecenie.Status[1] := TRUE;

                   //Obliczenie faktycznego czasu pracy (sekundy, zaokraglone)
                   #temp_diff_time := "DB_Zlecenia".Zlecenie["DB_Data".ZlecenieIndex[1]].Zlecenie."Time".Stanowisko2.EndTime - "DB_Zlecenia".Zlecenie["DB_Data".ZlecenieIndex[1]].Zlecenie."Time".Stanowisko2.StartTime;
                   "DB_Zlecenia".Zlecenie["DB_Data".ZlecenieIndex[1]].Zlecenie."Time".Stanowisko2.ActualTime := DINT_TO_INT((TIME_TO_DINT(#temp_diff_time) + 500) / 1000);
               END_IF;

               "DB_Data".ZlecenieIndex[1] := -1;
               "DB_Data".Stanowisko2.Commands.AbortProcess.State := 0;
               "DB_Data".Stanowisko2.Production.OrderNo := 0;
               "DB_Data".Stanowisko2.Production.ProductNo := 0;
               "DB_Data".Stanowisko2.Stats.Instruction := 1;
               "DB_Data".Stanowisko2.Production.State := 0;
           END_IF;

   END_CASE;
   IF "DB_Data".Stanowisko2.Commands.AbortProcess.State THEN
       "DB_Data".Stanowisko2.Production.State := 0;
       "DB_Data".Stanowisko2.Commands.AbortProcess.State := 0;

       IF "DB_Data".ZlecenieIndex[1] >= 0 THEN
           #temp_start_time := RD_LOC_T(OUT => "DB_Zlecenia".Zlecenie["DB_Data".ZlecenieIndex[1]].Zlecenie."Time".Stanowisko2.EndTime);
           "DB_Zlecenia".Zlecenie["DB_Data".ZlecenieIndex[1]].Zlecenie."Time".Stanowisko2.Abort := TRUE;

           //Status stanowiska 2 - praca zakonczona (przez abort)
           "DB_Zlecenia".Zlecenie["DB_Data".ZlecenieIndex[1]].Zlecenie.Status[1] := TRUE;

           //Obliczenie faktycznego czasu pracy (sekundy, zaokraglone)
           #temp_diff_time := "DB_Zlecenia".Zlecenie["DB_Data".ZlecenieIndex[1]].Zlecenie."Time".Stanowisko2.EndTime - "DB_Zlecenia".Zlecenie["DB_Data".ZlecenieIndex[1]].Zlecenie."Time".Stanowisko2.StartTime;
           "DB_Zlecenia".Zlecenie["DB_Data".ZlecenieIndex[1]].Zlecenie."Time".Stanowisko2.ActualTime := DINT_TO_INT((TIME_TO_DINT(#temp_diff_time) + 500) / 1000);
       END_IF;
       "DB_Data".Stanowisko2.Production.OrderNo := 0;
       "DB_Data".Stanowisko2.Production.ProductNo := 0;
       "DB_Data".Stanowisko2.Stats.Instruction := 1;

       "DB_Data".ZlecenieIndex[1] := -1;
   END_IF;
   IF "DB_Data".Stanowisko2.HMI.Clear THEN
       "DB_Data".Stanowisko2.Stats.DoneToday := 0;
       "DB_Data".Stanowisko2.HMI.Clear := 0;
   END_IF;
END_ORGANIZATION_BLOCK

ORGANIZATION_BLOCK "Stanowisko3"   // OB127, SCL, ProgramCycle
TITLE = "Main Program Sweep (Cycle)"
{ S7_Optimized_Access := 'TRUE' }
VERSION : 0.1
   VAR_INPUT
      Initial_Call : Bool;   // Initial call of this OB
      Remanence : Bool;   // =True, if remanent data are available
   END_VAR
   VAR_TEMP
      temp_start_time : Int;
      temp_taget_time : Int;
      i : Int;
      Czas_DTL : DTL;
      Status_Czasu : Int;
      Minuty : Int;
      Sekundy : Int;
      StrMin : String;
      StrSec : String;
      temp_diff_time : Time;
   END_VAR
BEGIN
   // ===================== STANOWISKO 3 =====================
   CASE "DB_Data".Stanowisko3.Production.State OF

       0:
           //Ustawienie przyciskow
           "DB_Data".Stanowisko3.Commands.AbortProcess.Enable := 0;
           "DB_Data".Stanowisko3.Commands.FInish.Enable := 0;
           "DB_Data".Stanowisko3.Commands.ReportFault.Enable := 0;

           //Wyzerowanie stanu przyciskow (na wypadek zaleglych klikniec)
           "DB_Data".Stanowisko3.Commands.FInish.State := 0;
           "DB_Data".Stanowisko3.Commands.ReportFault.State := 0;

           //Ustawienie awarii na 0
           "DB_Data".Stanowisko3.Commands.FaultReason.DamagedPart := 0;
           "DB_Data".Stanowisko3.Commands.FaultReason.MissingPart := 0;
           "DB_Data".Stanowisko3.Commands.FaultReason.Other := 0;
           "DB_Data".Stanowisko3.Commands.FaultReason.PalletFault := 0;
           "DB_Data".Stanowisko3.Commands.FaultReason.SensorFault := 0;
           "DB_Data".Stanowisko3.Commands.FaultReason.WrongInstruction := 0;

           //Reset czasu cyklu na wyswietlaczu
           "DB_Data".Stanowisko3."Time".RemainingStr := '00:00';

           //Reset numeru zlecenia
           "DB_Data".Stanowisko3.Production.OrderNo := 0;
           "DB_Data".Stanowisko3.Production.ProductNo := 0;

           //Zerowanie flagi ladowania
           "DB_Data".Stanowisko3.Stats.Loaded := 0;

           "DB_Data".Stanowisko3.Stats.Instruction := 1;

           //Zabezpieczenie indeksu bazy (ustawienie na wartość pustą)
           "DB_Data".ZlecenieIndex[2] := -1;
           "RFID_test".Bufor_Odczyt3[0] := 0;
           "RFID_test".Bufor_Odczyt3[1] := 0;
           "RFID_test".Bufor_Odczyt3[2] := 0;

           //Przejscie do montazu jezeli paletka jest aktywna i start klikniety
           IF "DB_Data".Stanowisko3.Sensors.PalletPresent THEN
               "DB_Data".Stanowisko3.Commands.Start.Enable := 1;
               IF "DB_Data".Stanowisko3.Commands.Start.State THEN
                   "DB_Data".Stanowisko3.Production.State := 1;
                   "DB_Data".Stanowisko3.Commands.Start.State := 0;
                   "DB_Data".Stanowisko3.MontazState := 0;
               END_IF;
           ELSE
               "DB_Data".Stanowisko3.Commands.Start.Enable := 0;
           END_IF;


       1:
           //Ustawienie przycisków
           "DB_Data".Stanowisko3.Commands.Start.Enable := 0;
           "DB_Data".Stanowisko3.Commands.AbortProcess.Enable := 1;
           "DB_Data".Stanowisko3.Commands.FInish.Enable := 1;
           "DB_Data".Stanowisko3.Commands.ReportFault.Enable := 1;

           CASE "DB_Data".Stanowisko3.MontazState OF
               0:
                   // Wysłanie komendy odczytu
                   "DB_Data".Stanowisko3.Sensors.RFID.CmdRead := TRUE;

                   // Pobranie danych z bufora
                   "DB_Data".Stanowisko3.Production.OrderNo := BYTE_TO_INT("RFID_test".Bufor_Odczyt3[0]);
                   "DB_Data".Stanowisko3.Stats.Instruction := BYTE_TO_INT("RFID_test".Bufor_Odczyt3[1]);
                   "DB_Data".Stanowisko3.Production.ProductNo := BYTE_TO_INT("RFID_test".Bufor_Odczyt3[2]);

                   // Szukanie TargetTime w tablicy zleceń
                   FOR #i := 0 TO 199 DO
                       IF "DB_Zlecenia".Zlecenie[#i].Zlecenie.ID = "DB_Data".Stanowisko3.Production.OrderNo AND "DB_Zlecenia".Zlecenie[#i].Zlecenie.PartNo = "DB_Data".Stanowisko3.Production.ProductNo THEN
                           "DB_Data".Stanowisko3."Time".RemainingSec := "DB_Zlecenia".Zlecenie[#i].Zlecenie."Time".Stanowisko3.TargetTime;
                           "DB_Data".ZlecenieIndex[2] := #i;
                           EXIT;
                       END_IF;
                   END_FOR;

                   IF "DB_Data".Stanowisko3.Production.OrderNo <> 0 THEN
                       "DB_Data".Stanowisko3.MontazState := 1;
                   END_IF;

               1:
                   "DB_Data".Stanowisko3."Time".Blink := FALSE;
                   "DB_Data".Stanowisko3.Sensors.RFID.CmdRead := FALSE;
                   #temp_start_time := RD_LOC_T(OUT => "DB_Zlecenia".Zlecenie["DB_Data".ZlecenieIndex[2]].Zlecenie."Time".Stanowisko3.StartTime);

                   "DB_Data".Stanowisko3.MontazState := 2;

               2:
                   #Status_Czasu := RD_SYS_T(OUT => #Czas_DTL);

                   IF #Czas_DTL.SECOND <> "DB_Data".Stanowisko3."Time".LastSec THEN
                       "DB_Data".Stanowisko3."Time".LastSec := #Czas_DTL.SECOND;

                       IF "DB_Data".Stanowisko3."Time".RemainingSec > 0 THEN
                           "DB_Data".Stanowisko3."Time".RemainingSec := "DB_Data".Stanowisko3."Time".RemainingSec - 1;
                       END_IF;

                       IF "DB_Data".Stanowisko3."Time".RemainingSec <= 0 THEN
                           "DB_Data".Stanowisko3."Time".Blink := NOT "DB_Data".Stanowisko3."Time".Blink;
                       END_IF;
                   END_IF;

                   #Minuty := "DB_Data".Stanowisko3."Time".RemainingSec / 60;
                   #Sekundy := "DB_Data".Stanowisko3."Time".RemainingSec MOD 60;

                   #StrMin := INT_TO_STRING(#Minuty);
                   #StrSec := INT_TO_STRING(#Sekundy);

                   #StrMin := RIGHT(IN := #StrMin, L := LEN(#StrMin) - 1);
                   #StrSec := RIGHT(IN := #StrSec, L := LEN(#StrSec) - 1);

                   IF #Minuty < 10 THEN
                       #StrMin := CONCAT(IN1 := '0', IN2 := #StrMin);
                   END_IF;
                   IF #Sekundy < 10 THEN
                       #StrSec := CONCAT(IN1 := '0', IN2 := #StrSec);
                   END_IF;

                   IF "DB_Data".Stanowisko3."Time".RemainingSec <= 0 AND "DB_Data".Stanowisko3."Time".Blink THEN
                       "DB_Data".Stanowisko3."Time".RemainingStr := '     ';
                   ELSE
                       "DB_Data".Stanowisko3."Time".RemainingStr := CONCAT(IN1 := #StrMin, IN2 := CONCAT(IN1 := ':', IN2 := #StrSec));
                   END_IF;

           END_CASE;

           //Przejscie do stanu awarii
           IF "DB_Data".Stanowisko3.Commands.ReportFault.State THEN
               "DB_Data".Stanowisko3.Production.State := 3;
               "DB_Data".Stanowisko3.Commands.ReportFault.State := 0;
           END_IF;

           //Przejscie do zakonczenia montazu
           IF "DB_Data".Stanowisko3.Commands.FInish.State THEN
               "DB_Data".Stanowisko3.Production.State := 2;
               "DB_Data".Stanowisko3.Commands.FInish.State := 0;
           END_IF;

       2:
           "DB_Data".Stanowisko3.Commands.Start.Enable := 0;
           "DB_Data".Stanowisko3.Commands.AbortProcess.Enable := 0;
           "DB_Data".Stanowisko3.Commands.FInish.Enable := 0;
           "DB_Data".Stanowisko3.Commands.ReportFault.Enable := 0;

           // Zapis tylko jeśli indeks został znaleziony
           IF "DB_Data".ZlecenieIndex[2] >= 0 THEN
               #temp_start_time := RD_LOC_T(OUT => "DB_Zlecenia".Zlecenie["DB_Data".ZlecenieIndex[2]].Zlecenie."Time".Stanowisko3.EndTime);

               //Status stanowiska 3 - praca zakonczona
               "DB_Zlecenia".Zlecenie["DB_Data".ZlecenieIndex[2]].Zlecenie.Status[2] := TRUE;

               //Obliczenie faktycznego czasu pracy (sekundy, zaokraglone)
               #temp_diff_time := "DB_Zlecenia".Zlecenie["DB_Data".ZlecenieIndex[2]].Zlecenie."Time".Stanowisko3.EndTime - "DB_Zlecenia".Zlecenie["DB_Data".ZlecenieIndex[2]].Zlecenie."Time".Stanowisko3.StartTime;
               "DB_Zlecenia".Zlecenie["DB_Data".ZlecenieIndex[2]].Zlecenie."Time".Stanowisko3.ActualTime := DINT_TO_INT((TIME_TO_DINT(#temp_diff_time) + 500) / 1000);
           END_IF;

           "DB_Data".Stanowisko3.Stats.DoneToday := "DB_Data".Stanowisko3.Stats.DoneToday + 1;
           "DB_Data".DoneAllTime[2] := "DB_Data".DoneAllTime[2] + 1;

           "DB_Data".ZlecenieIndex[2] := -1;
           "DB_Data".Stanowisko3.Production.State := 0;

       3:
           "DB_Data".Stanowisko3.Commands.Start.Enable := 0;
           "DB_Data".Stanowisko3.Commands.AbortProcess.Enable := 1;
           "DB_Data".Stanowisko3.Commands.FInish.Enable := 0;
           "DB_Data".Stanowisko3.Commands.ReportFault.Enable := 0;

           IF "DB_Data".ZlecenieIndex[2] >= 0 THEN
               "DB_Zlecenia".Zlecenie["DB_Data".ZlecenieIndex[2]].Zlecenie.Alarm.Stanowisko3 := "DB_Data".Stanowisko3.Commands.FaultReason;
           END_IF;

           IF "DB_Data".Stanowisko3.Commands.AbortProcess.State THEN
               IF "DB_Data".ZlecenieIndex[2] >= 0 THEN
                   #temp_start_time := RD_LOC_T(OUT => "DB_Zlecenia".Zlecenie["DB_Data".ZlecenieIndex[2]].Zlecenie."Time".Stanowisko3.EndTime);
                   "DB_Zlecenia".Zlecenie["DB_Data".ZlecenieIndex[2]].Zlecenie."Time".Stanowisko3.Abort := TRUE;

                   //Status stanowiska 3 - praca zakonczona (przez abort)
                   "DB_Zlecenia".Zlecenie["DB_Data".ZlecenieIndex[2]].Zlecenie.Status[2] := TRUE;

                   //Obliczenie faktycznego czasu pracy (sekundy, zaokraglone)
                   #temp_diff_time := "DB_Zlecenia".Zlecenie["DB_Data".ZlecenieIndex[2]].Zlecenie."Time".Stanowisko3.EndTime - "DB_Zlecenia".Zlecenie["DB_Data".ZlecenieIndex[2]].Zlecenie."Time".Stanowisko3.StartTime;
                   "DB_Zlecenia".Zlecenie["DB_Data".ZlecenieIndex[2]].Zlecenie."Time".Stanowisko3.ActualTime := DINT_TO_INT((TIME_TO_DINT(#temp_diff_time) + 500) / 1000);
               END_IF;

               "DB_Data".ZlecenieIndex[2] := -1;
               "DB_Data".Stanowisko3.Commands.AbortProcess.State := 0;
               "DB_Data".Stanowisko3.Production.OrderNo := 0;
               "DB_Data".Stanowisko3.Production.ProductNo := 0;
               "DB_Data".Stanowisko3.Stats.Instruction := 1;
               "DB_Data".Stanowisko3.Production.State := 0;
           END_IF;

   END_CASE;
   IF "DB_Data".Stanowisko3.Commands.AbortProcess.State THEN
       "DB_Data".Stanowisko3.Production.State := 0;
       "DB_Data".Stanowisko3.Commands.AbortProcess.State := 0;

       IF "DB_Data".ZlecenieIndex[2] >= 0 THEN
           #temp_start_time := RD_LOC_T(OUT => "DB_Zlecenia".Zlecenie["DB_Data".ZlecenieIndex[2]].Zlecenie."Time".Stanowisko3.EndTime);
           "DB_Zlecenia".Zlecenie["DB_Data".ZlecenieIndex[2]].Zlecenie."Time".Stanowisko3.Abort := TRUE;

           //Status stanowiska 3 - praca zakonczona (przez abort)
           "DB_Zlecenia".Zlecenie["DB_Data".ZlecenieIndex[2]].Zlecenie.Status[2] := TRUE;

           //Obliczenie faktycznego czasu pracy (sekundy, zaokraglone)
           #temp_diff_time := "DB_Zlecenia".Zlecenie["DB_Data".ZlecenieIndex[2]].Zlecenie."Time".Stanowisko3.EndTime - "DB_Zlecenia".Zlecenie["DB_Data".ZlecenieIndex[2]].Zlecenie."Time".Stanowisko3.StartTime;
           "DB_Zlecenia".Zlecenie["DB_Data".ZlecenieIndex[2]].Zlecenie."Time".Stanowisko3.ActualTime := DINT_TO_INT((TIME_TO_DINT(#temp_diff_time) + 500) / 1000);
       END_IF;
       "DB_Data".Stanowisko3.Production.OrderNo := 0;
       "DB_Data".Stanowisko3.Production.ProductNo := 0;
       "DB_Data".Stanowisko3.Stats.Instruction := 1;

       "DB_Data".ZlecenieIndex[2] := -1;
   END_IF;
   IF "DB_Data".Stanowisko3.HMI.Clear THEN
       "DB_Data".Stanowisko3.Stats.DoneToday := 0;
       "DB_Data".Stanowisko3.HMI.Clear := 0;
   END_IF;
END_ORGANIZATION_BLOCK

ORGANIZATION_BLOCK "StanowiskoQC"   // OB128, SCL, ProgramCycle
TITLE = "Main Program Sweep (Cycle)"
{ S7_Optimized_Access := 'TRUE' }
VERSION : 0.1
   VAR_INPUT
      Initial_Call : Bool;   // Initial call of this OB
      Remanence : Bool;   // =True, if remanent data are available
   END_VAR
   VAR_TEMP
      temp_start_time : Int;
      temp_taget_time : Int;
      i : Int;
      Czas_DTL : DTL;
      Status_Czasu : Int;
      Minuty : Int;
      Sekundy : Int;
      StrMin : String;
      StrSec : String;
      idx : Int;
      temp_diff_time : Time;
   END_VAR
BEGIN
   // ===================== STANOWISKO QC =====================
   CASE "DB_Data".StanowiskoQC.Production.State OF

       0:
           //Przyciski off
           "DB_Data".StanowiskoQC.Commands.OK.Enable := 0;
           "DB_Data".StanowiskoQC.Commands.NOK.Enable := 0;
           "DB_Data".StanowiskoQC.Commands.ReportFault.Enable := 0;

           //Reset stanu przyciskow
           "DB_Data".StanowiskoQC.Commands.OK.State := 0;
           "DB_Data".StanowiskoQC.Commands.NOK.State := 0;
           "DB_Data".StanowiskoQC.Commands.ReportFault.State := 0;

           //Reset awarii
           "DB_Data".StanowiskoQC.FaultReason.Camera := 0;
           "DB_Data".StanowiskoQC.FaultReason.NOK := 0;
           "DB_Data".StanowiskoQC.FaultReason.PalletFault := 0;
           "DB_Data".StanowiskoQC.FaultReason.RFID := 0;
           "DB_Data".StanowiskoQC.FaultReason.SensorFault := 0;
           "DB_Data".StanowiskoQC.FaultReason.Other := 0;

           //Reset czasu i kamery
           "DB_Data".StanowiskoQC."Time".RemainingStr := '00:00';
           "DB_Data".StanowiskoQC.HMI.CameraStatus := 0;

           //Reset zlecenia
           "DB_Data".StanowiskoQC.Production.OrderNo := 0;
           "DB_Data".StanowiskoQC.Production.ProductNo := 0;

           "DB_Data".StanowiskoQC.Stats.Loaded := 0;
           "DB_Data".StanowiskoQC.Stats.Instruction := 1;

           //Zabezpieczenie indeksu bazy
           "DB_Data".ZlecenieIndex[3] := -1;
           "RFID_test".Bufor_Odczyt4[0] := 0;
           "RFID_test".Bufor_Odczyt4[1] := 0;
           "RFID_test".Bufor_Odczyt4[2] := 0;

           //Start jezeli paletka obecna
           IF "DB_Data".StanowiskoQC.Sensors.PalletPresent THEN
               "DB_Data".StanowiskoQC.Commands.Start.Enable := 1;
               IF "DB_Data".StanowiskoQC.Commands.Start.State THEN
                   "DB_Data".StanowiskoQC.Production.State := 1;
                   "DB_Data".StanowiskoQC.Commands.Start.State := 0;
                   "DB_Data".StanowiskoQC.QualityState := 0;
               END_IF;
           ELSE
               "DB_Data".StanowiskoQC.Commands.Start.Enable := 0;
           END_IF;


       1:
           "DB_Data".StanowiskoQC.Commands.Start.Enable := 0;
           "DB_Data".StanowiskoQC.Commands.OK.Enable := 1;
           "DB_Data".StanowiskoQC.Commands.NOK.Enable := 1;
           "DB_Data".StanowiskoQC.Commands.ReportFault.Enable := 1;

           CASE "DB_Data".StanowiskoQC.QualityState OF
               0:
                   //Komenda odczytu RFID
                   "DB_Data".StanowiskoQC.Sensors.RFID.CmdRead := TRUE;

                   //Dane z bufora
                   "DB_Data".StanowiskoQC.Production.OrderNo := BYTE_TO_INT("RFID_test".Bufor_Odczyt4[0]);
                   "DB_Data".StanowiskoQC.Stats.Instruction := BYTE_TO_INT("RFID_test".Bufor_Odczyt4[1]);
                   "DB_Data".StanowiskoQC.Production.ProductNo := BYTE_TO_INT("RFID_test".Bufor_Odczyt4[2]);

                   //Szukanie TargetTime
                   FOR #i := 0 TO 199 DO
                       IF "DB_Zlecenia".Zlecenie[#i].Zlecenie.ID = "DB_Data".StanowiskoQC.Production.OrderNo AND "DB_Zlecenia".Zlecenie[#i].Zlecenie.PartNo = "DB_Data".StanowiskoQC.Production.ProductNo THEN
                           "DB_Data".StanowiskoQC."Time".RemainingSec := "DB_Zlecenia".Zlecenie[#i].Zlecenie."Time".StanowiskoQC.TargetTime;
                           "DB_Data".ZlecenieIndex[3] := #i;
                           EXIT;
                       END_IF;
                   END_FOR;

                   //Zlecenie inspekcji kamery
                   "DB_Data".StanowiskoQC.CameraControl.bZrobInspekcje := TRUE;

                   IF "DB_Data".StanowiskoQC.Production.OrderNo <> 0 THEN
                       "DB_Data".StanowiskoQC.Sensors.RFID.CmdRead := FALSE;
                       "DB_Data".StanowiskoQC.QualityState := 1;
                   END_IF;

               1:
                   "DB_Data".StanowiskoQC."Time".Blink := FALSE;
                   #temp_start_time := RD_LOC_T(OUT => "DB_Zlecenia".Zlecenie["DB_Data".ZlecenieIndex[3]].Zlecenie."Time".StanowiskoQC.StartTime);
                   "DB_Data".StanowiskoQC.QualityState := 2;

               2:
                   #Status_Czasu := RD_SYS_T(OUT => #Czas_DTL);

                   IF #Czas_DTL.SECOND <> "DB_Data".StanowiskoQC."Time".LastSec THEN
                       "DB_Data".StanowiskoQC."Time".LastSec := #Czas_DTL.SECOND;

                       IF "DB_Data".StanowiskoQC."Time".RemainingSec > 0 THEN
                           "DB_Data".StanowiskoQC."Time".RemainingSec := "DB_Data".StanowiskoQC."Time".RemainingSec - 1;
                       END_IF;

                       IF "DB_Data".StanowiskoQC."Time".RemainingSec <= 0 THEN
                           "DB_Data".StanowiskoQC."Time".Blink := NOT "DB_Data".StanowiskoQC."Time".Blink;
                       END_IF;
                   END_IF;

                   #Minuty := "DB_Data".StanowiskoQC."Time".RemainingSec / 60;
                   #Sekundy := "DB_Data".StanowiskoQC."Time".RemainingSec MOD 60;
                   #StrMin := INT_TO_STRING(#Minuty);
                   #StrSec := INT_TO_STRING(#Sekundy);
                   #StrMin := RIGHT(IN := #StrMin, L := LEN(#StrMin) - 1);
                   #StrSec := RIGHT(IN := #StrSec, L := LEN(#StrSec) - 1);

                   IF #Minuty < 10 THEN
                       #StrMin := CONCAT(IN1 := '0', IN2 := #StrMin);
                   END_IF;
                   IF #Sekundy < 10 THEN
                       #StrSec := CONCAT(IN1 := '0', IN2 := #StrSec);
                   END_IF;

                   IF "DB_Data".StanowiskoQC."Time".RemainingSec <= 0 AND "DB_Data".StanowiskoQC."Time".Blink THEN
                       "DB_Data".StanowiskoQC."Time".RemainingStr := '     ';
                   ELSE
                       "DB_Data".StanowiskoQC."Time".RemainingStr := CONCAT(IN1 := #StrMin, IN2 := CONCAT(IN1 := ':', IN2 := #StrSec));
                   END_IF;

           END_CASE;

           //Status kamery (zabezpieczony indeks; sprawdz offset -1 vs -2)
           #idx := "DB_Data".StanowiskoQC.Stats.Instruction - 2;
           IF #idx >= 0 AND #idx <= 5 THEN
               IF "DB_Data".StanowiskoQC.CameraControl.wynikOV[#idx] THEN
                   "DB_Data".StanowiskoQC.HMI.CameraStatus := 1;
               ELSE
                   "DB_Data".StanowiskoQC.HMI.CameraStatus := 2;
               END_IF;
           ELSE
               "DB_Data".StanowiskoQC.HMI.CameraStatus := 0;
           END_IF;

           //ReportFault -> stan awarii
           IF "DB_Data".StanowiskoQC.Commands.ReportFault.State THEN
               "DB_Data".StanowiskoQC.Production.State := 3;
               "DB_Data".StanowiskoQC.Commands.ReportFault.State := 0;
           END_IF;

           //OK -> zakonczenie (ReturnQC = TRUE)
           IF "DB_Data".StanowiskoQC.Commands.OK.State THEN
               "DB_Data".StanowiskoQC.Commands.OK.State := 0;
               "DB_Data".StanowiskoQC.Stats.PartsOK := "DB_Data".StanowiskoQC.Stats.PartsOK + 1;
               "DB_Data".StanowiskoQC.Stats.DoneToday := "DB_Data".StanowiskoQC.Stats.DoneToday + 1;
               "DB_Data".DoneAllTime[3] := "DB_Data".DoneAllTime[3] + 1;
               "DB_Zlecenia".Zlecenie["DB_Data".ZlecenieIndex[3]].Zlecenie.ReturnQC := TRUE;
               "DB_Data".StanowiskoQC.Production.State := 2;
           END_IF;

           //NOK -> zakonczenie (ReturnQC = FALSE)
           IF "DB_Data".StanowiskoQC.Commands.NOK.State THEN
               "DB_Data".StanowiskoQC.Commands.NOK.State := 0;
               "DB_Data".StanowiskoQC.Stats.PartsNOK := "DB_Data".StanowiskoQC.Stats.PartsNOK + 1;
               "DB_Data".StanowiskoQC.Stats.DoneToday := "DB_Data".StanowiskoQC.Stats.DoneToday + 1;
               "DB_Zlecenia".Zlecenie["DB_Data".ZlecenieIndex[3]].Zlecenie.ReturnQC := FALSE;
               "DB_Zlecenia".Zlecenie["DB_Data".ZlecenieIndex[3]].Zlecenie.NOK.Damage := "DB_Data".StanowiskoQC.Commands.NOK.Damage;
               "DB_Zlecenia".Zlecenie["DB_Data".ZlecenieIndex[3]].Zlecenie.NOK.NoBrick := "DB_Data".StanowiskoQC.Commands.NOK.NoBrick;
               "DB_Zlecenia".Zlecenie["DB_Data".ZlecenieIndex[3]].Zlecenie.NOK.Offset := "DB_Data".StanowiskoQC.Commands.NOK.Offset;
               "DB_Zlecenia".Zlecenie["DB_Data".ZlecenieIndex[3]].Zlecenie.NOK.Other := "DB_Data".StanowiskoQC.Commands.NOK.Other;
               "DB_Zlecenia".Zlecenie["DB_Data".ZlecenieIndex[3]].Zlecenie.NOK.WrongColour := "DB_Data".StanowiskoQC.Commands.NOK.WrongColour;
               "DB_Zlecenia".Zlecenie["DB_Data".ZlecenieIndex[3]].Zlecenie.NOK.WrongNumber := "DB_Data".StanowiskoQC.Commands.NOK.WrongNumber;
               "DB_Data".StanowiskoQC.Production.State := 2;
           END_IF;

       2:
           "DB_Data".StanowiskoQC.Commands.Start.Enable := 0;
           "DB_Data".StanowiskoQC.Commands.OK.Enable := 0;
           "DB_Data".StanowiskoQC.Commands.NOK.Enable := 0;
           "DB_Data".StanowiskoQC.Commands.ReportFault.Enable := 0;

           "DB_Data".StanowiskoQC.Stats.PartsPercent := (("DB_Data".StanowiskoQC.Stats.PartsOK * 100) / "DB_Data".StanowiskoQC.Stats.DoneToday);

           IF "DB_Data".ZlecenieIndex[3] >= 0 THEN
               #temp_start_time := RD_LOC_T(OUT => "DB_Zlecenia".Zlecenie["DB_Data".ZlecenieIndex[3]].Zlecenie."Time".StanowiskoQC.EndTime);

               //Status stanowiska QC - praca zakonczona
               "DB_Zlecenia".Zlecenie["DB_Data".ZlecenieIndex[3]].Zlecenie.Status[3] := TRUE;

               //Obliczenie faktycznego czasu pracy (sekundy, zaokraglone)
               #temp_diff_time := "DB_Zlecenia".Zlecenie["DB_Data".ZlecenieIndex[3]].Zlecenie."Time".StanowiskoQC.EndTime - "DB_Zlecenia".Zlecenie["DB_Data".ZlecenieIndex[3]].Zlecenie."Time".StanowiskoQC.StartTime;
               "DB_Zlecenia".Zlecenie["DB_Data".ZlecenieIndex[3]].Zlecenie."Time".StanowiskoQC.ActualTime := DINT_TO_INT((TIME_TO_DINT(#temp_diff_time) + 500) / 1000);
           END_IF;

           "DB_Data".ZlecenieIndex[3] := -1;
           "DB_Data".StanowiskoQC.Production.State := 0;

       3:
           "DB_Data".StanowiskoQC.Commands.Start.Enable := 0;
           "DB_Data".StanowiskoQC.Commands.OK.Enable := 1;
           "DB_Data".StanowiskoQC.Commands.NOK.Enable := 1;
           "DB_Data".StanowiskoQC.Commands.ReportFault.Enable := 0;

           IF "DB_Data".ZlecenieIndex[3] >= 0 THEN
               "DB_Zlecenia".Zlecenie["DB_Data".ZlecenieIndex[3]].Zlecenie.Alarm.StanowieskoQC := "DB_Data".StanowiskoQC.FaultReason;
           END_IF;

           IF "DB_Data".StanowiskoQC.Commands.OK.State OR "DB_Data".StanowiskoQC.Commands.NOK.State THEN
               IF "DB_Data".ZlecenieIndex[3] >= 0 THEN
                   #temp_start_time := RD_LOC_T(OUT => "DB_Zlecenia".Zlecenie["DB_Data".ZlecenieIndex[3]].Zlecenie."Time".StanowiskoQC.EndTime);

                   //Status stanowiska QC - praca zakonczona (z trybu awarii)
                   "DB_Zlecenia".Zlecenie["DB_Data".ZlecenieIndex[3]].Zlecenie.Status[3] := TRUE;

                   //Obliczenie faktycznego czasu pracy (sekundy, zaokraglone)
                   #temp_diff_time := "DB_Zlecenia".Zlecenie["DB_Data".ZlecenieIndex[3]].Zlecenie."Time".StanowiskoQC.EndTime - "DB_Zlecenia".Zlecenie["DB_Data".ZlecenieIndex[3]].Zlecenie."Time".StanowiskoQC.StartTime;
                   "DB_Zlecenia".Zlecenie["DB_Data".ZlecenieIndex[3]].Zlecenie."Time".StanowiskoQC.ActualTime := DINT_TO_INT((TIME_TO_DINT(#temp_diff_time) + 500) / 1000);

                   "DB_Zlecenia".Zlecenie["DB_Data".ZlecenieIndex[3]].Zlecenie.Alarm.StanowieskoQC := "DB_Data".StanowiskoQC.FaultReason;

                   "DB_Zlecenia".Zlecenie["DB_Data".ZlecenieIndex[3]].Zlecenie.NOK.Damage := "DB_Data".StanowiskoQC.Commands.NOK.Damage;
                   "DB_Zlecenia".Zlecenie["DB_Data".ZlecenieIndex[3]].Zlecenie.NOK.NoBrick := "DB_Data".StanowiskoQC.Commands.NOK.NoBrick;
                   "DB_Zlecenia".Zlecenie["DB_Data".ZlecenieIndex[3]].Zlecenie.NOK.Offset := "DB_Data".StanowiskoQC.Commands.NOK.Offset;
                   "DB_Zlecenia".Zlecenie["DB_Data".ZlecenieIndex[3]].Zlecenie.NOK.Other := "DB_Data".StanowiskoQC.Commands.NOK.Other;
                   "DB_Zlecenia".Zlecenie["DB_Data".ZlecenieIndex[3]].Zlecenie.NOK.WrongColour := "DB_Data".StanowiskoQC.Commands.NOK.WrongColour;
                   "DB_Zlecenia".Zlecenie["DB_Data".ZlecenieIndex[3]].Zlecenie.NOK.WrongNumber := "DB_Data".StanowiskoQC.Commands.NOK.WrongNumber;
               END_IF;

               "DB_Data".ZlecenieIndex[3] := -1;
               "DB_Data".StanowiskoQC.Production.OrderNo := 0;
               "DB_Data".StanowiskoQC.Production.ProductNo := 0;
               "DB_Data".StanowiskoQC.Stats.Instruction := 1;
               "DB_Data".StanowiskoQC.Production.State := 0;
               "DB_Data".StanowiskoQC.Commands.OK.State := 0;
               "DB_Data".StanowiskoQC.Commands.NOK.State := 0;
           END_IF;

   END_CASE;
   IF "DB_Data".StanowiskoQC.HMI.Clear THEN
       "DB_Data".StanowiskoQC.Stats.DoneToday := 0;
       "DB_Data".StanowiskoQC.Stats.PartsNOK := 0;
       "DB_Data".StanowiskoQC.Stats.PartsOK := 0;
       "DB_Data".StanowiskoQC.Stats.PartsPercent := 0;
       "DB_Data".StanowiskoQC.HMI.Clear := 0;
   END_IF;
END_ORGANIZATION_BLOCK

ORGANIZATION_BLOCK "ResetZleceń"   // OB129, SCL, ProgramCycle
TITLE = "Main Program Sweep (Cycle)"
{ S7_Optimized_Access := 'TRUE' }
VERSION : 0.1
   VAR_INPUT
      Initial_Call : Bool;   // Initial call of this OB
      Remanence : Bool;   // =True, if remanent data are available
   END_VAR
   VAR_TEMP
      i : Int;
   END_VAR
BEGIN
   IF "DB_Zlecenia".ResetZlecen THEN

       //Reszet tablicy
       FOR #i := 0 TO 199 DO
           "DB_Zlecenia".Zlecenie[#i] := "DB_Zlecenia".PusteZlecenie;
       END_FOR;

       //Reset nastepnego zlecenia
       "DB_Zlecenia".NastepneZlecenie := "DB_Zlecenia".PusteZlecenie;

       //Reset stanu resetu po skonczonym zadaniu
       "DB_Zlecenia".ResetZlecen := FALSE;

       //Reset do stanu zero stanowisk
       "DB_Data".Stanowisko1.Production.State := 0;
       "DB_Data".Stanowisko2.Production.State := 0;
       "DB_Data".Stanowisko3.Production.State := 0;
       "DB_Data".StanowiskoQC.Production.State := 0;
   END_IF;
END_ORGANIZATION_BLOCK